GLOBALCONSTANTS AID_OLA (* Output list object attribute ids *)
  (* Standard: 61499-1; Description: Copyright (c) 2023 HR Agrartechnik GmbH This program and the accompanying materials are made available under the terms of the Eclipse Public License 2.0 which is available at https://www.eclipse.org/legal/epl-2.0/ SPDX-License-Identifier: EPL-2.0 *)
  (* Version 1.0, 2026-06-20, Franz Höpfinger, HR Agrartechnik GmbH *)
  PACKAGE isobus::UT::Q::const::AID;
  VAR_GLOBAL CONSTANT
    WIDTH : USINT := USINT#1; (* 1: AID_OLA_WIDTH - Width in pixels. *)
    HEIGHT : USINT := USINT#2; (* 2: AID_OLA_HEIGHT - Height in pixels. *)
    VARIABLE_REF : USINT := USINT#3; (* 3: AID_OLA_VARIABLE_REF - Object ID of a Number Variable object. *)
    VALUE : USINT := USINT#4; (* 4: AID_OLA_VALUE (read-only) - Selected list index (0 to 254), or 255 if no item is chosen. *)
  END_VAR
END_GLOBALCONSTANTS
